// TIA Portal V18 export
// export: Created 2025-12-01T12:38:53.9181367Z, ExportSetting None, DisplayName Totally Integrated Automation Portal, DisplayVersion V18 Update 5, DisplayName TIA Portal Openness, DisplayVersion V18 Update 5, DisplayName TIA Portal Teamcenter Gateway, DisplayVersion V18, DisplayName TIA Portal Version Control Interface, DisplayVersion V18, DisplayName STEP 7 Professional, DisplayVersion V18 Update 5, DisplayName STEP 7 Safety, DisplayVersion V18, DisplayName WinCC Professional, DisplayVersion V18 Update 5
FUNCTION "ST10_PartData" : Void   // FC1500, SCL
{ S7_Optimized_Access := 'TRUE' }
// stored: SetENOAutomatically false
   VAR_INPUT
      iSysMode : "RCS_SysComInterface_V1";
   END_VAR
   VAR_TEMP
      idex : Int;
   END_VAR
BEGIN
END_FUNCTION
